// TIA Portal V21 export
DATA_BLOCK "PHTRe"   // DB41
{ S7_Optimized_Access := 'TRUE' }
// stored: AutoNumber false, MemoryReserve 100
   VAR
      PhtLinePrintText : Array[0..10] of String[40];
      PhtLinePrint1 : String[40];
      RE : Array[0..20] of Bool;
   END_VAR
BEGIN
   PhtLinePrintText[1] := 'PRESSURIZE STARTED';
   PhtLinePrintText[2] := 'STABILIZE STARTED';
   PhtLinePrintText[3] := 'PRESSURE HOLD STARTED';
   PhtLinePrintText[4] := 'PRESSURE RELEASE STARTED';
   PhtLinePrintText[5] := 'CYCLE PAUSED';
   PhtLinePrintText[6] := 'PHT OVER';
END_DATA_BLOCK
